KUKA KRL data list: up23.dat

&ACCESS RV7
&REL 383
&COMMENT VW380 Kleben
&PARAM DISKPATH = KRC:\R1\UPs
&PARAM TEMPLATE = C:\KRC\Roboter\Template\upvorgabe
&PARAM TPVW_VERSION = 8.1.8
&PARAM EDITMASK = Up999[1-999]
DEFDAT UP23
; FOLD ;%{H} %MKUKATPVW
; ENDFOLD
; interface to basic routines
 EXT  BAS (BAS_COMMAND  :IN,REAL  :IN )
; interface to VW-standard routines
EXT VW (VW_COMMAND:IN, BOOL: IN, REAL:IN, REAL:IN, REAL:IN, REAL:IN, BOOL :IN, E6POS :IN )
; interface to VW_USER - Call
EXT  VW_USER (VW_USER_CMD :IN,INT :IN,REAL  :IN,REAL  :IN,REAL  :IN,REAL  :IN,REAL  :IN,REAL  :IN,BOOL  :IN )
EXT  VW_USR_R (VW_USER_CMD :IN,INT :IN,REAL  :IN,REAL  :IN,REAL  :IN,REAL  :IN,REAL  :IN,REAL  :IN,BOOL  :IN )
EXT  IBGN (IBGN_COMMAND  :IN,BOOL  :IN,REAL  :IN,REAL  :IN,BOOL  :IN,E6POS  :OUT )
; interface select routine
EXTFCT INT  SELECT (SUBTYPE  :IN,INT  :IN,BOOL  :IN,ARI_TYP  :IN,INT  :IN,BOOL_TYP  :IN,INT  :IN,BOOL  :IN)
INT VW_NEXT_FREE = 60
INT VW_NFREE_SPS = 60
INT VW_MAX_SPS = 160
DECL VW_MPARA_TYP P1_D = {TOOL_NO 13,BASE_NO 0,VB 100,VE 0,ACC 100,TRG_TIME 0,MOVE_TYPE #PTP_MOTION}
DECL E6POS P1 = {X 1999.569, Y -2389.745, Z 1521.284, A 90.00037, B -0.000257676, C 29.99883, S 2, T 42 , E1 0.0, E2 0.0, E3 0.0, E4 0.0, E5 0.0, E6 0.0}
DECL VW_MPARA_TYP P2_D = {TOOL_NO 13,BASE_NO 3,VB 100,VE 100,ACC 100,TRG_TIME 0,MOVE_TYPE #PTP_MOTION}
DECL E6POS P2 = {X 1909.465, Y -388.8534, Z -1133.924, A -98.69143, B 29.4809, C -7.535059, S 2, T 42 , E1 0.0, E2 0.0, E3 0.0, E4 0.0, E5 0.0, E6 0.0}
DECL VW_MPARA_TYP P3_D = {TOOL_NO 13,BASE_NO 3,VB 100,VE 100,ACC 100,TRG_TIME 0,MOVE_TYPE #PTP_MOTION}
DECL E6POS P3 = {X 2928.199, Y 803.7011, Z 1239.667, A -30.55688, B -19.96261, C 100.3486, S 6, T 50 , E1 0.0, E2 0.0, E3 0.0, E4 0.0, E5 0.0, E6 0.0}
DECL VW_MPARA_TYP P4_D = {TOOL_NO 13,BASE_NO 3,VB 100,VE 100,ACC 100,TRG_TIME 0,MOVE_TYPE #PTP_MOTION}
DECL E6POS P4 = {X 2511.858, Y 770.7318, Z 944.9971, A -45.01979, B -4.578051, C 100.0725, S 6, T 50 , E1 0.0, E2 0.0, E3 0.0, E4 0.0, E5 0.0, E6 0.0}
DECL VW_MPARA_TYP P5_D = {TOOL_NO 13,BASE_NO 3,VB 100,VE 100,ACC 100,TRG_TIME 0,MOVE_TYPE #PTP_MOTION}
DECL E6POS P5 = {X 2431.337, Y 643.8981, Z 921.5394, A -49.35415, B -3.824125, C 100.2685, S 6, T 50 , E1 0.0, E2 0.0, E3 0.0, E4 0.0, E5 0.0, E6 0.0}
DECL VW_MPARA_TYP P6_D = {TOOL_NO 13,BASE_NO 3,VB 100,VE 100,ACC 100,TRG_TIME 0,MOVE_TYPE #PTP_MOTION}
DECL E6POS P6 = {X 2443.099, Y 616.2974, Z 935.1517, A -49.43446, B -2.70017, C 109.405, S 6, T 50 , E1 0.0, E2 0.0, E3 0.0, E4 0.0, E5 0.0, E6 0.0}
DECL VW_MPARA_TYP P7_D = {TOOL_NO 13,BASE_NO 3,VB 150,VE 25,ACC 50,TRG_TIME 0,MOVE_TYPE #GLUE_MOTION}
DECL E6POS P7 = {X 2449.753, Y 600.6858, Z 942.8785, A -49.47981, B -2.064372, C 114.5727, S 6, T 50 , E1 0.0, E2 0.0, E3 0.0, E4 0.0, E5 0.0, E6 0.0}
DECL VW_MPARA_TYP P8_D = {TOOL_NO 13,BASE_NO 3,VB 150,VE 25,ACC 50,TRG_TIME 0,MOVE_TYPE #GLUE_MOTION}
DECL E6POS P8 = {X 2453.1, Y 596.5966, Z 941.7529, A -49.47982, B -2.064378, C 114.5727, S 6, T 50 , E1 0.0, E2 0.0, E3 0.0, E4 0.0, E5 0.0, E6 0.0}
DECL VW_MPARA_TYP P9_D = {TOOL_NO 13,BASE_NO 3,VB 150,VE 25,ACC 50,TRG_TIME 0,MOVE_TYPE #GLUE_MOTION}
DECL E6POS P9 = {X 2472.68, Y 608.1747, Z 913.2568, A -49.47984, B -2.06452, C 114.5729, S 6, T 50 , E1 0.0, E2 0.0, E3 0.0, E4 0.0, E5 0.0, E6 0.0}
DECL VW_MPARA_TYP P10_D = {TOOL_NO 13,BASE_NO 3,VB 150,VE 25,ACC 50,TRG_TIME 0,MOVE_TYPE #GLUE_MOTION}
DECL E6POS P10 = {X 2491.583, Y 620.0996, Z 882.9735, A -49.47963, B -2.064557, C 114.5726, S 6, T 50 , E1 0.0, E2 0.0, E3 0.0, E4 0.0, E5 0.0, E6 0.0}
DECL VW_MPARA_TYP P11_D = {TOOL_NO 13,BASE_NO 3,VB 150,VE 25,ACC 50,TRG_TIME 0,MOVE_TYPE #GLUE_MOTION}
DECL E6POS P11 = {X 2496.983, Y 625.7777, Z 872.1993, A -48.20971, B 0.7132434, C 114.56, S 6, T 50 , E1 0.0, E2 0.0, E3 0.0, E4 0.0, E5 0.0, E6 0.0}
DECL VW_MPARA_TYP P12_D = {TOOL_NO 13,BASE_NO 3,VB 150,VE 25,ACC 50,TRG_TIME 0,MOVE_TYPE #GLUE_MOTION}
DECL E6POS P12 = {X 2500.767, Y 629.8958, Z 863.1186, A -47.17876, B 2.966972, C 114.5911, S 6, T 50 , E1 0.0, E2 0.0, E3 0.0, E4 0.0, E5 0.0, E6 0.0}
DECL VW_MPARA_TYP P13_D = {TOOL_NO 13,BASE_NO 3,VB 150,VE 25,ACC 50,TRG_TIME 0,MOVE_TYPE #GLUE_MOTION}
DECL E6POS P13 = {X 2505.107, Y 634.7009, Z 851.3597, A -44.13681, B 5.91533, C 114.707, S 6, T 50 , E1 0.0, E2 0.0, E3 0.0, E4 0.0, E5 0.0, E6 0.0}
DECL VW_MPARA_TYP P14_D = {TOOL_NO 13,BASE_NO 3,VB 150,VE 25,ACC 50,TRG_TIME 0,MOVE_TYPE #GLUE_MOTION}
DECL E6POS P14 = {X 2507.774, Y 642.0746, Z 838.9906, A -40.81743, B 9.075095, C 115.0107, S 6, T 50 , E1 0.0, E2 0.0, E3 0.0, E4 0.0, E5 0.0, E6 0.0}
DECL VW_MPARA_TYP P15_D = {TOOL_NO 13,BASE_NO 3,VB 150,VE 25,ACC 50,TRG_TIME 0,MOVE_TYPE #GLUE_MOTION}
DECL E6POS P15 = {X 2508.523, Y 650.1994, Z 823.6599, A -35.97059, B 13.53225, C 115.7778, S 6, T 50 , E1 0.0, E2 0.0, E3 0.0, E4 0.0, E5 0.0, E6 0.0}
DECL VW_MPARA_TYP P16_D = {TOOL_NO 13,BASE_NO 3,VB 150,VE 25,ACC 50,TRG_TIME 0,MOVE_TYPE #GLUE_MOTION}
DECL E6POS P16 = {X 2507.231, Y 654.6443, Z 813.4005, A -33.12129, B 16.04003, C 116.3994, S 6, T 50 , E1 0.0, E2 0.0, E3 0.0, E4 0.0, E5 0.0, E6 0.0}
DECL VW_MPARA_TYP P17_D = {TOOL_NO 13,BASE_NO 3,VB 150,VE 25,ACC 50,TRG_TIME 0,MOVE_TYPE #GLUE_MOTION}
DECL E6POS P17 = {X 2500.057, Y 665.0558, Z 792.556, A -31.43494, B 26.98918, C 116.7515, S 6, T 50 , E1 0.0, E2 0.0, E3 0.0, E4 0.0, E5 0.0, E6 0.0}
DECL VW_MPARA_TYP P18_D = {TOOL_NO 13,BASE_NO 3,VB 150,VE 25,ACC 50,TRG_TIME 0,MOVE_TYPE #GLUE_MOTION}
DECL E6POS P18 = {X 2494.341, Y 671.3528, Z 779.7806, A -31.00417, B 30.09447, C 117.6911, S 6, T 50 , E1 0.0, E2 0.0, E3 0.0, E4 0.0, E5 0.0, E6 0.0}
DECL VW_MPARA_TYP P19_D = {TOOL_NO 13,BASE_NO 3,VB 150,VE 25,ACC 50,TRG_TIME 0,MOVE_TYPE #GLUE_MOTION}
DECL E6POS P19 = {X 2465.187, Y 693.8577, Z 733.2496, A -26.24541, B 33.9754, C 121.9999, S 6, T 50 , E1 0.0, E2 0.0, E3 0.0, E4 0.0, E5 0.0, E6 0.0}
DECL VW_MPARA_TYP P20_D = {TOOL_NO 13,BASE_NO 3,VB 150,VE 25,ACC 50,TRG_TIME 0,MOVE_TYPE #GLUE_MOTION}
DECL E6POS P20 = {X 2434.635, Y 716.3539, Z 688.3223, A -23.79696, B 32.92177, C 122.8941, S 6, T 50 , E1 0.0, E2 0.0, E3 0.0, E4 0.0, E5 0.0, E6 0.0}
DECL VW_MPARA_TYP P21_D = {TOOL_NO 13,BASE_NO 3,VB 150,VE 25,ACC 50,TRG_TIME 0,MOVE_TYPE #GLUE_MOTION}
DECL E6POS P21 = {X 2426.139, Y 723.631, Z 674.5562, A -23.47899, B 32.488, C 122.909, S 6, T 50 , E1 0.0, E2 0.0, E3 0.0, E4 0.0, E5 0.0, E6 0.0}
DECL VW_MPARA_TYP P22_D = {TOOL_NO 13,BASE_NO 3,VB 150,VE 25,ACC 50,TRG_TIME 0,MOVE_TYPE #GLUE_MOTION}
DECL E6POS P22 = {X 2408.827, Y 711.7422, Z 652.1298, A -23.328, B 32.815, C 123.088, S 6, T 50 , E1 0.0, E2 0.0, E3 0.0, E4 0.0, E5 0.0, E6 0.0}
DECL VW_MPARA_TYP P23_D = {TOOL_NO 13,BASE_NO 3,VB 150,VE 25,ACC 50,TRG_TIME 0,MOVE_TYPE #GLUE_MOTION}
DECL E6POS P23 = {X 2409.355, Y 733.4708, Z 648.8415, A -23.328, B 32.815, C 123.088, S 6, T 50 , E1 0.0, E2 0.0, E3 0.0, E4 0.0, E5 0.0, E6 0.0}
DECL VW_MPARA_TYP P24_D = {TOOL_NO 13,BASE_NO 3,VB 150,VE 25,ACC 50,TRG_TIME 0,MOVE_TYPE #GLUE_MOTION}
DECL E6POS P24 = {X 2409.664, Y 744.9827, Z 647.1776, A -23.328, B 32.815, C 123.088, S 6, T 50 , E1 0.0, E2 0.0, E3 0.0, E4 0.0, E5 0.0, E6 0.0}
DECL VW_MPARA_TYP P25_D = {TOOL_NO 13,BASE_NO 3,VB 150,VE 25,ACC 50,TRG_TIME 0,MOVE_TYPE #GLUE_MOTION}
DECL E6POS P25 = {X 2405.577, Y 733.4557, Z 644.3956, A -23.32801, B 32.81512, C 123.0879, S 6, T 50 , E1 0.0, E2 0.0, E3 0.0, E4 0.0, E5 0.0, E6 0.0}
DECL VW_MPARA_TYP P26_D = {TOOL_NO 13,BASE_NO 3,VB 150,VE 25,ACC 50,TRG_TIME 0,MOVE_TYPE #GLUE_MOTION}
DECL E6POS P26 = {X 2401.917, Y 711.067, Z 642.0864, A -23.328, B 32.815, C 123.088, S 6, T 50 , E1 0.0, E2 0.0, E3 0.0, E4 0.0, E5 0.0, E6 0.0}
DECL VW_MPARA_TYP P27_D = {TOOL_NO 13,BASE_NO 3,VB 150,VE 25,ACC 50,TRG_TIME 0,MOVE_TYPE #GLUE_MOTION}
DECL E6POS P27 = {X 2391.126, Y 719.16, Z 625.0737, A -23.03106, B 32.95296, C 123.2769, S 6, T 50 , E1 0.0, E2 0.0, E3 0.0, E4 0.0, E5 0.0, E6 0.0}
DECL VW_MPARA_TYP P28_D = {TOOL_NO 13,BASE_NO 3,VB 150,VE 25,ACC 50,TRG_TIME 0,MOVE_TYPE #GLUE_MOTION}
DECL E6POS P28 = {X 2382.983, Y 727.0417, Z 611.4378, A -22.92001, B 33.426, C 123.4899, S 6, T 50 , E1 0.0, E2 0.0, E3 0.0, E4 0.0, E5 0.0, E6 0.0}
DECL VW_MPARA_TYP P29_D = {TOOL_NO 13,BASE_NO 3,VB 150,VE 25,ACC 50,TRG_TIME 0,MOVE_TYPE #GLUE_MOTION}
DECL E6POS P29 = {X 2377.674, Y 732.3444, Z 603.7584, A -22.86905, B 33.58679, C 123.5681, S 6, T 50 , E1 0.0, E2 0.0, E3 0.0, E4 0.0, E5 0.0, E6 0.0}
DECL VW_MPARA_TYP P30_D = {TOOL_NO 13,BASE_NO 3,VB 150,VE 25,ACC 50,TRG_TIME 0,MOVE_TYPE #GLUE_MOTION}
DECL E6POS P30 = {X 2356.512, Y 725.9248, Z 590.2668, A -22.843, B 33.665, C 123.6081, S 6, T 50 , E1 0.0, E2 0.0, E3 0.0, E4 0.0, E5 0.0, E6 0.0}
DECL VW_MPARA_TYP P31_D = {TOOL_NO 13,BASE_NO 3,VB 150,VE 25,ACC 50,TRG_TIME 0,MOVE_TYPE #GLUE_MOTION}
DECL E6POS P31 = {X 2385.707, Y 727.1175, Z 618.7888, A -14.94098, B 34.45401, C 131.374, S 6, T 50 , E1 0.0, E2 0.0, E3 0.0, E4 0.0, E5 0.0, E6 0.0}
DECL VW_MPARA_TYP P32_D = {TOOL_NO 13,BASE_NO 3,VB 150,VE 25,ACC 50,TRG_TIME 0,MOVE_TYPE #GLUE_MOTION}
DECL E6POS P32 = {X 2387.704, Y 732.1568, Z 617.4284, A -11.78399, B 34.69952, C 137.1981, S 6, T 50 , E1 0.0, E2 0.0, E3 0.0, E4 0.0, E5 0.0, E6 0.0}
DECL VW_MPARA_TYP P33_D = {TOOL_NO 13,BASE_NO 3,VB 150,VE 25,ACC 50,TRG_TIME 0,MOVE_TYPE #GLUE_MOTION}
DECL E6POS P33 = {X 2392.277, Y 756.3744, Z 620.7583, A -4.964964, B 34.94344, C 149.777, S 6, T 50 , E1 0.0, E2 0.0, E3 0.0, E4 0.0, E5 0.0, E6 0.0}
DECL VW_MPARA_TYP P34_D = {TOOL_NO 13,BASE_NO 3,VB 150,VE 25,ACC 50,TRG_TIME 0,MOVE_TYPE #GLUE_MOTION}
DECL E6POS P34 = {X 2394.421, Y 772.3488, Z 625.1818, A -4.964949, B 34.944, C 149.777, S 6, T 50 , E1 0.0, E2 0.0, E3 0.0, E4 0.0, E5 0.0, E6 0.0}
DECL VW_MPARA_TYP P35_D = {TOOL_NO 13,BASE_NO 3,VB 100,VE 100,ACC 100,TRG_TIME 0,MOVE_TYPE #PTP_MOTION}
DECL E6POS P35 = {X 2386.288, Y 758.8298, Z 633.9037, A -17.97797, B 37.71602, C 140.119, S 6, T 50 , E1 0.0, E2 0.0, E3 0.0, E4 0.0, E5 0.0, E6 0.0}
DECL VW_MPARA_TYP P36_D = {TOOL_NO 13,BASE_NO 3,VB 100,VE 10,ACC 100,TRG_TIME 0,MOVE_TYPE #PTP_MOTION}
DECL E6POS P36 = {X 2397.542, Y 733.978, Z 655.4952, A -41.22901, B 35.51999, C 119.145, S 6, T 50 , E1 0.0, E2 0.0, E3 0.0, E4 0.0, E5 0.0, E6 0.0}
DECL VW_MPARA_TYP P37_D = {TOOL_NO 13,BASE_NO 3,VB 100,VE 10,ACC 100,TRG_TIME 0,MOVE_TYPE #PTP_MOTION}
DECL E6POS P37 = {X 2347.888, Y 708.1067, Z 641.9673, A -60.89103, B 37.16293, C 107.051, S 6, T 50 , E1 0.0, E2 0.0, E3 0.0, E4 0.0, E5 0.0, E6 0.0}
DECL VW_MPARA_TYP P38_D = {TOOL_NO 13,BASE_NO 3,VB 100,VE 10,ACC 100,TRG_TIME 0,MOVE_TYPE #PTP_MOTION}
DECL E6POS P38 = {X 2341.394, Y 742.1302, Z 686.652, A -75.86099, B 30.78704, C 94.30801, S 6, T 50 , E1 0.0, E2 0.0, E3 0.0, E4 0.0, E5 0.0, E6 0.0}
DECL VW_MPARA_TYP P39_D = {TOOL_NO 13,BASE_NO 3,VB 100,VE 10,ACC 100,TRG_TIME 0,MOVE_TYPE #PTP_MOTION}
DECL E6POS P39 = {X 2404.216, Y 733.9532, Z 723.4583, A -96.06801, B 12.34904, C 74.80399, S 6, T 50 , E1 0.0, E2 0.0, E3 0.0, E4 0.0, E5 0.0, E6 0.0}
DECL VW_MPARA_TYP P40_D = {TOOL_NO 13,BASE_NO 3,VB 100,VE 100,ACC 100,TRG_TIME 0,MOVE_TYPE #PTP_MOTION}
DECL E6POS P40 = {X 2418.986, Y 714.1864, Z 724.8347, A -113.678, B 0.2610787, C 67.61499, S 6, T 50 , E1 0.0, E2 0.0, E3 0.0, E4 0.0, E5 0.0, E6 0.0}
DECL VW_MPARA_TYP P41_D = {TOOL_NO 13,BASE_NO 3,VB 150,VE 25,ACC 50,TRG_TIME 0,MOVE_TYPE #GLUE_MOTION}
DECL E6POS P41 = {X 2410.794, Y 687.6442, Z 724.3491, A -119.0371, B -3.530925, C 66.15321, S 6, T 50 , E1 0.0, E2 0.0, E3 0.0, E4 0.0, E5 0.0, E6 0.0}
DECL VW_MPARA_TYP P42_D = {TOOL_NO 13,BASE_NO 3,VB 150,VE 25,ACC 50,TRG_TIME 0,MOVE_TYPE #GLUE_MOTION}
DECL E6POS P42 = {X 2423.018, Y 684.6837, Z 736.8874, A -119.0371, B -3.530925, C 66.15321, S 6, T 50 , E1 0.0, E2 0.0, E3 0.0, E4 0.0, E5 0.0, E6 0.0}
DECL VW_MPARA_TYP P43_D = {TOOL_NO 13,BASE_NO 3,VB 150,VE 25,ACC 50,TRG_TIME 0,MOVE_TYPE #GLUE_MOTION}
DECL E6POS P43 = {X 2439.956, Y 677.6878, Z 757.7448, A -123.339, B -4.299047, C 65.99896, S 6, T 50 , E1 0.0, E2 0.0, E3 0.0, E4 0.0, E5 0.0, E6 0.0}
DECL VW_MPARA_TYP P44_D = {TOOL_NO 13,BASE_NO 3,VB 150,VE 25,ACC 50,TRG_TIME 0,MOVE_TYPE #GLUE_MOTION}
DECL E6POS P44 = {X 2456.76, Y 668.2476, Z 780.0774, A -128.553, B -5.195, C 65.89001, S 6, T 50 , E1 0.0, E2 0.0, E3 0.0, E4 0.0, E5 0.0, E6 0.0}
DECL VW_MPARA_TYP P45_D = {TOOL_NO 13,BASE_NO 3,VB 150,VE 25,ACC 50,TRG_TIME 0,MOVE_TYPE #GLUE_MOTION}
DECL E6POS P45 = {X 2468.137, Y 661.0607, Z 797.2104, A -129.9465, B -0.1839993, C 65.78481, S 6, T 50 , E1 0.0, E2 0.0, E3 0.0, E4 0.0, E5 0.0, E6 0.0}
DECL VW_MPARA_TYP P46_D = {TOOL_NO 13,BASE_NO 3,VB 150,VE 25,ACC 50,TRG_TIME 0,MOVE_TYPE #GLUE_MOTION}
DECL E6POS P46 = {X 2474.421, Y 655.5244, Z 811.5954, A -129.7418, B 6.30159, C 69.83949, S 6, T 50 , E1 0.0, E2 0.0, E3 0.0, E4 0.0, E5 0.0, E6 0.0}
DECL VW_MPARA_TYP P47_D = {TOOL_NO 13,BASE_NO 3,VB 150,VE 25,ACC 50,TRG_TIME 0,MOVE_TYPE #GLUE_MOTION}
DECL E6POS P47 = {X 2478.229, Y 651.2855, Z 823.6866, A -127.7067, B 16.88149, C 72.66247, S 6, T 50 , E1 0.0, E2 0.0, E3 0.0, E4 0.0, E5 0.0, E6 0.0}
DECL VW_MPARA_TYP P48_D = {TOOL_NO 13,BASE_NO 3,VB 150,VE 25,ACC 50,TRG_TIME 0,MOVE_TYPE #GLUE_MOTION}
DECL E6POS P48 = {X 2479.326, Y 647.9109, Z 833.2495, A -124.8824, B 25.35215, C 74.90589, S 6, T 50 , E1 0.0, E2 0.0, E3 0.0, E4 0.0, E5 0.0, E6 0.0}
DECL VW_MPARA_TYP P49_D = {TOOL_NO 13,BASE_NO 3,VB 150,VE 25,ACC 50,TRG_TIME 0,MOVE_TYPE #GLUE_MOTION}
DECL E6POS P49 = {X 2477.65, Y 644.3282, Z 842.7652, A -121.175, B 31.42147, C 75.4511, S 6, T 50 , E1 0.0, E2 0.0, E3 0.0, E4 0.0, E5 0.0, E6 0.0}
DECL VW_MPARA_TYP P50_D = {TOOL_NO 13,BASE_NO 3,VB 150,VE 25,ACC 50,TRG_TIME 0,MOVE_TYPE #GLUE_MOTION}
DECL E6POS P50 = {X 2475.876, Y 640.2809, Z 852.188, A -124.9084, B 31.56287, C 72.11004, S 6, T 50 , E1 0.0, E2 0.0, E3 0.0, E4 0.0, E5 0.0, E6 0.0}
DECL VW_MPARA_TYP P51_D = {TOOL_NO 13,BASE_NO 3,VB 150,VE 25,ACC 50,TRG_TIME 0,MOVE_TYPE #GLUE_MOTION}
DECL E6POS P51 = {X 2469.288, Y 632.0369, Z 869.6974, A -123.0707, B 35.75963, C 70.07247, S 6, T 50 , E1 0.0, E2 0.0, E3 0.0, E4 0.0, E5 0.0, E6 0.0}
DECL VW_MPARA_TYP P52_D = {TOOL_NO 13,BASE_NO 3,VB 150,VE 25,ACC 50,TRG_TIME 0,MOVE_TYPE #GLUE_MOTION}
DECL E6POS P52 = {X 2458.774, Y 624.0023, Z 886.495, A -120.629, B 42.38057, C 70.97793, S 6, T 50 , E1 0.0, E2 0.0, E3 0.0, E4 0.0, E5 0.0, E6 0.0}
DECL VW_MPARA_TYP P53_D = {TOOL_NO 13,BASE_NO 3,VB 150,VE 25,ACC 50,TRG_TIME 0,MOVE_TYPE #GLUE_MOTION}
DECL E6POS P53 = {X 2449.388, Y 617.5876, Z 902.3852, A -123.3, B 43.07133, C 72.12955, S 6, T 50 , E1 0.0, E2 0.0, E3 0.0, E4 0.0, E5 0.0, E6 0.0}
DECL VW_MPARA_TYP P54_D = {TOOL_NO 13,BASE_NO 3,VB 150,VE 25,ACC 50,TRG_TIME 0,MOVE_TYPE #GLUE_MOTION}
DECL E6POS P54 = {X 2435.586, Y 608.6146, Z 922.6822, A -123.3, B 43.07133, C 72.12955, S 6, T 50 , E1 0.0, E2 0.0, E3 0.0, E4 0.0, E5 0.0, E6 0.0}
DECL VW_MPARA_TYP P55_D = {TOOL_NO 13,BASE_NO 3,VB 100,VE 100,ACC 100,TRG_TIME 0,MOVE_TYPE #PTP_MOTION}
DECL E6POS P55 = {X 2441.472, Y 650.2891, Z 966.1577, A -123.3, B 43.07133, C 72.12955, S 6, T 50 , E1 0.0, E2 0.0, E3 0.0, E4 0.0, E5 0.0, E6 0.0}
DECL VW_MPARA_TYP P56_D = {TOOL_NO 13,BASE_NO 3,VB 100,VE 100,ACC 100,TRG_TIME 0,MOVE_TYPE #PTP_MOTION}
DECL E6POS P56 = {X 2571.239, Y 822.9655, Z 828.0203, A -88.32969, B 27.47893, C 86.27706, S 6, T 50 , E1 0.0, E2 0.0, E3 0.0, E4 0.0, E5 0.0, E6 0.0}
DECL VW_MPARA_TYP P57_D = {TOOL_NO 13,BASE_NO 3,VB 100,VE 100,ACC 100,TRG_TIME 0,MOVE_TYPE #PTP_MOTION}
DECL E6POS P57 = {X 2773.542, Y 654.4924, Z 476.3365, A -57.9698, B 25.85835, C 100.1762, S 6, T 50 , E1 0.0, E2 0.0, E3 0.0, E4 0.0, E5 0.0, E6 0.0}
DECL VW_MPARA_TYP P58_D = {TOOL_NO 13,BASE_NO 3,VB 100,VE 100,ACC 100,TRG_TIME 0,MOVE_TYPE #PTP_MOTION}
DECL E6POS P58 = {X 3690.665, Y 1776.87, Z -416.2481, A 3.101173, B 37.14202, C 103.1819, S 6, T 50 , E1 0.0, E2 0.0, E3 0.0, E4 0.0, E5 0.0, E6 0.0}
DECL VW_MPARA_TYP P59_D = {TOOL_NO 13,BASE_NO 0,VB 100,VE 0,ACC 100,TRG_TIME 0,MOVE_TYPE #PTP_MOTION}
DECL E6POS P59 = {X 1999.569, Y -2389.746, Z 1521.285, A 90.00037, B -0.000254692, C 29.99883, S 2, T 42 , E1 0.0, E2 0.0, E3 0.0, E4 0.0, E5 0.0, E6 0.0}
ENDDAT
